SUBAPPLICATION INI_IN_AND_STORE_AR2_TO_REAL (* INI Laden und Speichern (wie INI_IN_AND_STORE_AR2), zusaetzlich per AR_R_TO_REAL auf einen plain-REAL-OutputVar konvertiert - fuer InputVars auf Ziel-FBs, die einen echten REAL-Parameter statt eines AR-Adapter-Sockets erwarten (z.B. CTRL_PID_AR.KP/TN/TV). *)
  (* Standard: 61499-2; Description: Copyright (c) 2026 Meisterschulen am Ostbahnhof This program and the accompanying materials are made available under the terms of the Eclipse Public License 2.0 which is available at https://www.eclipse.org/legal/epl-2.0/ SPDX-License-Identifier: EPL-2.0 *)
  (* Version 1.0, 2026-09-15, Franz Höpfinger, Meisterschulen am Ostbahnhof, initial implementation - aus Aufnahme_Automatik.SUB herausgeloest (dort 3x identisch fuer KP/TN/TV verdrahtet: INI_IN_AND_STORE_AR2 + AR_R_TO_REAL). INI_IN_AND_STORE_AR2.VALUEO (AR) -> AR_R_TO_REAL.AR_IN -> VALUE (REAL-OutputVar). *)
  PACKAGE MyLib::sys;
  IMPORT isobus::UT::Q::const::IDs::ID_NULL;
  IMPORT logiBUS::utils::conversion::phys::NumericObjectPool_S;
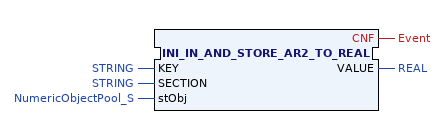
  EVENT_OUTPUT
    CNF; (* Confirmation - feuert wenn ein (neuer oder initial geladener) Wert vorliegt. An einen REQ-Eingang eines Ziel-FB anschliessen (z.B. CTRL_PID_AR.REQ), damit dieser den frischen Wert sofort uebernimmt, statt auf den naechsten eigenen Adapter-Trigger zu warten. *)
  END_EVENT
  VAR_INPUT
    KEY : STRING; (* Key name. *)
    SECTION : STRING; (* Section name. *)
    stObj : logiBUS::utils::conversion::phys::NumericObjectPool_S := (u16ObjId := ID_NULL, r32Scale := 1.0, i32Offset := 0, u8Decimals := 0);
  END_VAR
  VAR_OUTPUT
    VALUE : REAL; (* Persistierter/geladener Wert, plain REAL (nicht AR-Adapter) - fuer InputVars auf Ziel-FBs, die einen echten REAL-Parameter erwarten. *)
  END_VAR
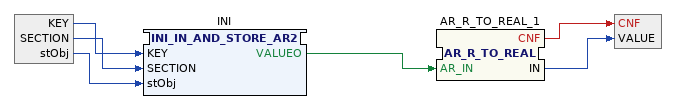
  FBS
    AR_R_TO_REAL_1 : adapter::conversion::unidirectional::AR_R_TO_REAL;
  END_FBS
  SUBAPPS
    INI : MyLib::sys::INI_IN_AND_STORE_AR2;
  END_SUBAPPS
  EVENT_CONNECTIONS
    AR_R_TO_REAL_1.CNF TO CNF;
  END_CONNECTIONS
  DATA_CONNECTIONS
    KEY TO INI.KEY;
    SECTION TO INI.SECTION;
    stObj TO INI.stObj;
    AR_R_TO_REAL_1.IN TO VALUE;
  END_CONNECTIONS
  ADAPTER_CONNECTIONS
    INI.VALUEO TO AR_R_TO_REAL_1.AR_IN;
  END_CONNECTIONS
END_SUBAPPLICATION
